Fanuc KAREL source: kt00307.KL

-- PROVISIONAL review KL for V940-1; original PC SHA256 4d7ca6f1f30252e4d3e377d510b9c887c3e9d76385c3bc96ba233923ce3dfe87
-- Incomplete behavior may be omitted. Consult companion uncertainty JSON. Do not deploy.
PROGRAM KT00307
%NOLOCKGROUP
VAR
  I2 : INTEGER
  OUT : BOOLEAN
-- UNRESOLVED_DECL H1 type=002017
BEGIN
  -- V9_ZERO_TABLE_METADATA_HINT layout=0001; no indexed target words; source/name/runtime held
  -- UNRESOLVED_PC offsets 5-19; opcodes 2E,22,9D,33,B4
  -- UNRESOLVED_PC offsets 24-35; opcodes 2E,23
  -- UNRESOLVED_PC offsets 40-62; opcodes 22,9D,33,B3,21,58,23
  -- UNRESOLVED_PC offsets 67-71; opcodes 7F
END KT00307
